{attribute 'pack_mode' := '2'}
TYPE ST_XTS_TRANSPORT_STATE :
STRUCT
  State         : E_XTS_TRANSPORT_STATE;  // combined value of state and result(e_progress); (hint: extract state value by mod division)
  Check         : E_XTS_TRANSPORT_CHECK;

  XpuState      : ST_XPU_STATE;
  XpuInfo       : ST_XPU_INFO;
  GroupInfo     : ST_GROUP_INFO; 
END_STRUCT
END_TYPE

(* stored: Version 1.1.0.1
   DUT ST_XTS_TRANSPORT_STATE: Id {3e744e9d-3ef1-45b6-9c08-c979549e1166} *)
